ABB RAPID module: f527d16c.mod

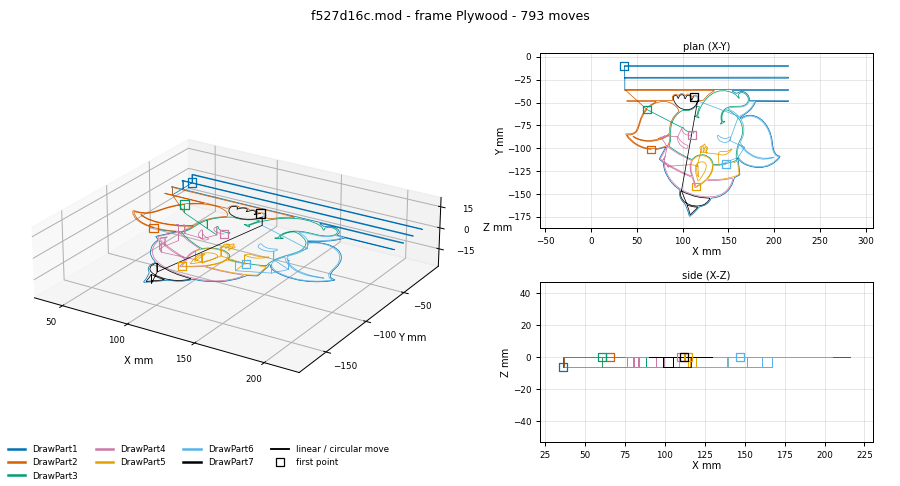
[picture p0: tool path of f527d16c.mod in frame Plywood, 793 of 795 moves have a stored position in this frame; points joined in program order, loops and branches not executed]
MODULE ImageDraw
  ! Generated 2026-10-07 09:04 for ABB GoFa CRB 15000-5/0.95: 26 strokes
  ! Page 250 x 180 mm. Work object Plywood: Z points DOWN, so pen-up is -Z and the tool uses orientation [1,0,0,0].
  ! Uses the tool 'tcp' and work object 'Plywood' that already exist on the controller.
  CONST robtarget pOrigin:=[[0,0,0],[1,0,0,0],[0,0,0,0],[9E9,9E9,9E9,9E9,9E9,9E9]];
  CONST jointtarget jHome:=[[0,0,0,0,30,0],[9E9,9E9,9E9,9E9,9E9,9E9]];
  CONST speeddata vTravel:=[250,200,5000,1000];

  PROC DrawImage()
    SingArea\Wrist;
    ConfL\Off;
    ConfJ\Off;
    MoveAbsJ jHome\NoEOffs,vTravel,fine,tcp;
    DrawPart1;
    DrawPart2;
    DrawPart3;
    DrawPart4;
    DrawPart5;
    DrawPart6;
    DrawPart7;
    MoveAbsJ jHome\NoEOffs,vTravel,fine,tcp;
  ENDPROC

  PROC DrawPart1()
    MoveL Offs(pOrigin,36.30,-10.13,-6.00),vTravel,z5,tcp\WObj:=Plywood;
    MoveL Offs(pOrigin,36.30,-10.13,-0.00),v60,z0,tcp\WObj:=Plywood;
    MoveL Offs(pOrigin,37.06,-9.56,-0.00),v40,z0,tcp\WObj:=Plywood;
    MoveL Offs(pOrigin,215.03,-9.56,-0.00),v40,z0,tcp\WObj:=Plywood;
    MoveL Offs(pOrigin,215.98,-9.94,-0.00),v40,z0,tcp\WObj:=Plywood;
    MoveL Offs(pOrigin,215.60,-10.51,-0.00),v40,z0,tcp\WObj:=Plywood;
    MoveL Offs(pOrigin,38.96,-10.70,-0.00),v40,z0,tcp\WObj:=Plywood;
    MoveL Offs(pOrigin,36.68,-10.51,-0.00),v40,z0,tcp\WObj:=Plywood;
    MoveL Offs(pOrigin,36.30,-10.13,-0.00),v40,fine,tcp\WObj:=Plywood;
    MoveL Offs(pOrigin,36.30,-10.13,-6.00),v60,z5,tcp\WObj:=Plywood;
    MoveL Offs(pOrigin,36.87,-22.47,-6.00),vTravel,z5,tcp\WObj:=Plywood;
    MoveL Offs(pOrigin,36.87,-22.47,-0.00),v60,z0,tcp\WObj:=Plywood;
    MoveL Offs(pOrigin,213.13,-22.28,-0.00),v40,z0,tcp\WObj:=Plywood;
    MoveL Offs(pOrigin,215.60,-22.47,-0.00),v40,z0,tcp\WObj:=Plywood;
    MoveL Offs(pOrigin,215.98,-22.85,-0.00),v40,z0,tcp\WObj:=Plywood;
    MoveL Offs(pOrigin,215.41,-23.42,-0.00),v40,z0,tcp\WObj:=Plywood;
    MoveL Offs(pOrigin,36.68,-23.42,-0.00),v40,z0,tcp\WObj:=Plywood;
    MoveL Offs(pOrigin,36.30,-23.04,-0.00),v40,z0,tcp\WObj:=Plywood;
    MoveL Offs(pOrigin,36.87,-22.47,-0.00),v40,fine,tcp\WObj:=Plywood;
    MoveL Offs(pOrigin,36.87,-22.47,-6.00),v60,z5,tcp\WObj:=Plywood;
    MoveL Offs(pOrigin,36.87,-35.77,-6.00),vTravel,z5,tcp\WObj:=Plywood;
    MoveL Offs(pOrigin,36.87,-35.77,-0.00),v60,z0,tcp\WObj:=Plywood;
    MoveL Offs(pOrigin,107.34,-35.96,-0.00),v40,z0,tcp\WObj:=Plywood;
    MoveL Offs(pOrigin,150.64,-35.58,-0.00),v40,z0,tcp\WObj:=Plywood;
    MoveL Offs(pOrigin,215.41,-35.77,-0.00),v40,z0,tcp\WObj:=Plywood;
    MoveL Offs(pOrigin,215.98,-36.15,-0.00),v40,z0,tcp\WObj:=Plywood;
    MoveL Offs(pOrigin,215.60,-36.72,-0.00),v40,z0,tcp\WObj:=Plywood;
    MoveL Offs(pOrigin,206.87,-36.91,-0.00),v40,z0,tcp\WObj:=Plywood;
    MoveL Offs(pOrigin,167.36,-36.72,-0.00),v40,z0,tcp\WObj:=Plywood;
    MoveL Offs(pOrigin,155.20,-36.91,-0.00),v40,z0,tcp\WObj:=Plywood;
    MoveL Offs(pOrigin,154.25,-37.16,-0.00),v40,z0,tcp\WObj:=Plywood;
    MoveL Offs(pOrigin,154.63,-37.73,-0.00),v40,z0,tcp\WObj:=Plywood;
    MoveL Offs(pOrigin,158.81,-40.01,-0.00),v40,z0,tcp\WObj:=Plywood;
    MoveL Offs(pOrigin,159.76,-39.44,-0.00),v40,z0,tcp\WObj:=Plywood;
    MoveL Offs(pOrigin,160.52,-39.44,-0.00),v40,z0,tcp\WObj:=Plywood;
    MoveL Offs(pOrigin,163.37,-37.86,-0.00),v40,z0,tcp\WObj:=Plywood;
    MoveL Offs(pOrigin,165.46,-37.86,-0.00),v40,z0,tcp\WObj:=Plywood;
    MoveL Offs(pOrigin,167.36,-38.37,-0.00),v40,z0,tcp\WObj:=Plywood;
    MoveL Offs(pOrigin,169.07,-39.25,-0.00),v40,z0,tcp\WObj:=Plywood;
    MoveL Offs(pOrigin,171.79,-42.23,-0.00),v40,z0,tcp\WObj:=Plywood;
    MoveL Offs(pOrigin,172.87,-44.70,-0.00),v40,z0,tcp\WObj:=Plywood;
    MoveL Offs(pOrigin,172.93,-47.55,-0.00),v40,z0,tcp\WObj:=Plywood;
    MoveL Offs(pOrigin,173.63,-47.93,-0.00),v40,z0,tcp\WObj:=Plywood;
    MoveL Offs(pOrigin,215.92,-48.12,-0.00),v40,z0,tcp\WObj:=Plywood;
    MoveL Offs(pOrigin,215.79,-48.62,-0.00),v40,z0,tcp\WObj:=Plywood;
    MoveL Offs(pOrigin,214.65,-48.88,-0.00),v40,z0,tcp\WObj:=Plywood;
    MoveL Offs(pOrigin,179.89,-48.81,-0.00),v40,z0,tcp\WObj:=Plywood;
    MoveL Offs(pOrigin,177.93,-53.06,-0.00),v40,z0,tcp\WObj:=Plywood;
    MoveL Offs(pOrigin,174.58,-57.61,-0.00),v40,z0,tcp\WObj:=Plywood;
    MoveL Offs(pOrigin,170.78,-61.03,-0.00),v40,z0,tcp\WObj:=Plywood;
    MoveL Offs(pOrigin,162.48,-66.54,-0.00),v40,z0,tcp\WObj:=Plywood;
    MoveL Offs(pOrigin,163.18,-67.49,-0.00),v40,z0,tcp\WObj:=Plywood;
    MoveL Offs(pOrigin,167.36,-65.15,-0.00),v40,z0,tcp\WObj:=Plywood;
    MoveL Offs(pOrigin,169.45,-64.45,-0.00),v40,z0,tcp\WObj:=Plywood;
    MoveL Offs(pOrigin,172.87,-63.88,-0.00),v40,z0,tcp\WObj:=Plywood;
    MoveL Offs(pOrigin,176.66,-64.07,-0.00),v40,z0,tcp\WObj:=Plywood;
    MoveL Offs(pOrigin,180.84,-65.34,-0.00),v40,z0,tcp\WObj:=Plywood;
    MoveL Offs(pOrigin,183.12,-66.48,-0.00),v40,z0,tcp\WObj:=Plywood;
    MoveL Offs(pOrigin,186.73,-69.01,-0.00),v40,z0,tcp\WObj:=Plywood;
    MoveL Offs(pOrigin,190.72,-73.38,-0.00),v40,z0,tcp\WObj:=Plywood;
    MoveL Offs(pOrigin,193.25,-77.37,-0.00),v40,z0,tcp\WObj:=Plywood;
    MoveL Offs(pOrigin,195.34,-81.74,-0.00),v40,z0,tcp\WObj:=Plywood;
    MoveL Offs(pOrigin,197.56,-89.34,-0.00),v40,z0,tcp\WObj:=Plywood;
    MoveL Offs(pOrigin,198.51,-97.31,-0.00),v40,z0,tcp\WObj:=Plywood;
    MoveL Offs(pOrigin,199.96,-103.20,-0.00),v40,z0,tcp\WObj:=Plywood;
    MoveL Offs(pOrigin,202.12,-106.62,-0.00),v40,z0,tcp\WObj:=Plywood;
    MoveL Offs(pOrigin,204.21,-108.01,-0.00),v40,z0,tcp\WObj:=Plywood;
    MoveL Offs(pOrigin,206.30,-108.58,-0.00),v40,z0,tcp\WObj:=Plywood;
    MoveL Offs(pOrigin,206.36,-109.47,-0.00),v40,z0,tcp\WObj:=Plywood;
    MoveL Offs(pOrigin,203.07,-113.46,-0.00),v40,z0,tcp\WObj:=Plywood;
    MoveL Offs(pOrigin,198.13,-117.13,-0.00),v40,z0,tcp\WObj:=Plywood;
    MoveL Offs(pOrigin,193.38,-119.41,-0.00),v40,z0,tcp\WObj:=Plywood;
    MoveL Offs(pOrigin,187.11,-120.87,-0.00),v40,z0,tcp\WObj:=Plywood;
    MoveL Offs(pOrigin,180.27,-120.87,-0.00),v40,z0,tcp\WObj:=Plywood;
    MoveL Offs(pOrigin,176.28,-120.30,-0.00),v40,z0,tcp\WObj:=Plywood;
    MoveL Offs(pOrigin,171.16,-118.84,-0.00),v40,z0,tcp\WObj:=Plywood;
    MoveL Offs(pOrigin,167.36,-117.13,-0.00),v40,z0,tcp\WObj:=Plywood;
    MoveL Offs(pOrigin,164.89,-115.55,-0.00),v40,z0,tcp\WObj:=Plywood;
    MoveL Offs(pOrigin,162.42,-113.27,-0.00),v40,z0,tcp\WObj:=Plywood;
    MoveL Offs(pOrigin,160.52,-110.61,-0.00),v40,z0,tcp\WObj:=Plywood;
    MoveL Offs(pOrigin,160.14,-110.48,-0.00),v40,z0,tcp\WObj:=Plywood;
    MoveL Offs(pOrigin,159.95,-111.37,-0.00),v40,z0,tcp\WObj:=Plywood;
    MoveL Offs(pOrigin,160.90,-113.84,-0.00),v40,z0,tcp\WObj:=Plywood;
    MoveL Offs(pOrigin,162.61,-128.46,-0.00),v40,z0,tcp\WObj:=Plywood;
    MoveL Offs(pOrigin,162.23,-129.22,-0.00),v40,z0,tcp\WObj:=Plywood;
    MoveL Offs(pOrigin,156.72,-132.07,-0.00),v40,z0,tcp\WObj:=Plywood;
    MoveL Offs(pOrigin,154.12,-139.67,-0.00),v40,z0,tcp\WObj:=Plywood;
    MoveL Offs(pOrigin,150.26,-145.75,-0.00),v40,z0,tcp\WObj:=Plywood;
    MoveL Offs(pOrigin,147.03,-148.79,-0.00),v40,z0,tcp\WObj:=Plywood;
    MoveL Offs(pOrigin,141.53,-152.14,-0.00),v40,z0,tcp\WObj:=Plywood;
    MoveL Offs(pOrigin,136.78,-153.73,-0.00),v40,z0,tcp\WObj:=Plywood;
    MoveL Offs(pOrigin,131.27,-154.55,-0.00),v40,z0,tcp\WObj:=Plywood;
    MoveL Offs(pOrigin,129.94,-157.15,-0.00),v40,z0,tcp\WObj:=Plywood;
    MoveL Offs(pOrigin,127.28,-160.18,-0.00),v40,z0,tcp\WObj:=Plywood;
    MoveL Offs(pOrigin,124.24,-162.21,-0.00),v40,z0,tcp\WObj:=Plywood;
    MoveL Offs(pOrigin,118.35,-164.17,-0.00),v40,z0,tcp\WObj:=Plywood;
    MoveL Offs(pOrigin,111.51,-171.39,-0.00),v40,z0,tcp\WObj:=Plywood;
    MoveL Offs(pOrigin,107.91,-174.37,-0.00),v40,z0,tcp\WObj:=Plywood;
    MoveL Offs(pOrigin,107.27,-173.86,-0.00),v40,z0,tcp\WObj:=Plywood;
    MoveL Offs(pOrigin,105.88,-168.92,-0.00),v40,z0,tcp\WObj:=Plywood;
    MoveL Offs(pOrigin,103.09,-161.89,-0.00),v40,z0,tcp\WObj:=Plywood;
    MoveL Offs(pOrigin,102.21,-160.37,-0.00),v40,z0,tcp\WObj:=Plywood;
    MoveL Offs(pOrigin,99.17,-156.96,-0.00),v40,z0,tcp\WObj:=Plywood;
    MoveL Offs(pOrigin,97.58,-154.11,-0.00),v40,z0,tcp\WObj:=Plywood;
    MoveL Offs(pOrigin,96.70,-150.88,-0.00),v40,z0,tcp\WObj:=Plywood;
    MoveL Offs(pOrigin,96.70,-148.41,-0.00),v40,z0,tcp\WObj:=Plywood;
    MoveL Offs(pOrigin,97.20,-145.75,-0.00),v40,z0,tcp\WObj:=Plywood;
    MoveL Offs(pOrigin,91.95,-141.57,-0.00),v40,z0,tcp\WObj:=Plywood;
    MoveL Offs(pOrigin,88.15,-137.77,-0.00),v40,z0,tcp\WObj:=Plywood;
    MoveL Offs(pOrigin,85.30,-133.97,-0.00),v40,z0,tcp\WObj:=Plywood;
    MoveL Offs(pOrigin,81.82,-127.70,-0.00),v40,z0,tcp\WObj:=Plywood;
    MoveL Offs(pOrigin,80.49,-124.28,-0.00),v40,z0,tcp\WObj:=Plywood;
    MoveL Offs(pOrigin,79.41,-120.11,-0.00),v40,z0,tcp\WObj:=Plywood;
    MoveL Offs(pOrigin,78.91,-115.55,-0.00),v40,z0,tcp\WObj:=Plywood;
    MoveL Offs(pOrigin,74.73,-112.13,-0.00),v40,z0,tcp\WObj:=Plywood;
    MoveL Offs(pOrigin,75.17,-110.42,-0.00),v40,z0,tcp\WObj:=Plywood;
    MoveL Offs(pOrigin,81.63,-98.83,-0.00),v40,z0,tcp\WObj:=Plywood;
    MoveL Offs(pOrigin,81.12,-98.64,-0.00),v40,z0,tcp\WObj:=Plywood;
    MoveL Offs(pOrigin,75.04,-100.54,-0.00),v40,z0,tcp\WObj:=Plywood;
    MoveL Offs(pOrigin,70.30,-101.30,-0.00),v40,z0,tcp\WObj:=Plywood;
  ENDPROC

  PROC DrawPart2()
    MoveL Offs(pOrigin,65.55,-101.30,-0.00),v40,z0,tcp\WObj:=Plywood;
    MoveL Offs(pOrigin,57.95,-99.97,-0.00),v40,z0,tcp\WObj:=Plywood;
    MoveL Offs(pOrigin,51.68,-97.57,-0.00),v40,z0,tcp\WObj:=Plywood;
    MoveL Offs(pOrigin,46.17,-94.08,-0.00),v40,z0,tcp\WObj:=Plywood;
    MoveL Offs(pOrigin,41.23,-89.53,-0.00),v40,z0,tcp\WObj:=Plywood;
    MoveL Offs(pOrigin,37.94,-84.97,-0.00),v40,z0,tcp\WObj:=Plywood;
    MoveL Offs(pOrigin,38.39,-84.21,-0.00),v40,z0,tcp\WObj:=Plywood;
    MoveL Offs(pOrigin,43.13,-84.21,-0.00),v40,z0,tcp\WObj:=Plywood;
    MoveL Offs(pOrigin,46.36,-83.32,-0.00),v40,z0,tcp\WObj:=Plywood;
    MoveL Offs(pOrigin,47.50,-82.69,-0.00),v40,z0,tcp\WObj:=Plywood;
    MoveL Offs(pOrigin,49.21,-80.98,-0.00),v40,z0,tcp\WObj:=Plywood;
    MoveL Offs(pOrigin,51.18,-76.80,-0.00),v40,z0,tcp\WObj:=Plywood;
    MoveL Offs(pOrigin,54.28,-66.92,-0.00),v40,z0,tcp\WObj:=Plywood;
    MoveL Offs(pOrigin,56.56,-62.17,-0.00),v40,z0,tcp\WObj:=Plywood;
    MoveL Offs(pOrigin,58.14,-59.70,-0.00),v40,z0,tcp\WObj:=Plywood;
    MoveL Offs(pOrigin,61.56,-55.53,-0.00),v40,z0,tcp\WObj:=Plywood;
    MoveL Offs(pOrigin,64.60,-52.87,-0.00),v40,z0,tcp\WObj:=Plywood;
    MoveL Offs(pOrigin,71.12,-49.07,-0.00),v40,z0,tcp\WObj:=Plywood;
    MoveL Offs(pOrigin,70.68,-48.69,-0.00),v40,z0,tcp\WObj:=Plywood;
    MoveL Offs(pOrigin,39.34,-48.69,-0.00),v40,z0,tcp\WObj:=Plywood;
    MoveL Offs(pOrigin,38.96,-48.31,-0.00),v40,z0,tcp\WObj:=Plywood;
    MoveL Offs(pOrigin,39.15,-47.99,-0.00),v40,z0,tcp\WObj:=Plywood;
    MoveL Offs(pOrigin,88.72,-47.93,-0.00),v40,z0,tcp\WObj:=Plywood;
    MoveL Offs(pOrigin,89.29,-47.36,-0.00),v40,z0,tcp\WObj:=Plywood;
    MoveL Offs(pOrigin,88.72,-43.75,-0.00),v40,z0,tcp\WObj:=Plywood;
    MoveL Offs(pOrigin,90.05,-41.85,-0.00),v40,z0,tcp\WObj:=Plywood;
    MoveL Offs(pOrigin,91.95,-40.96,-0.00),v40,z0,tcp\WObj:=Plywood;
    MoveL Offs(pOrigin,93.66,-41.09,-0.00),v40,z0,tcp\WObj:=Plywood;
    MoveL Offs(pOrigin,95.37,-42.29,-0.00),v40,z0,tcp\WObj:=Plywood;
    MoveL Offs(pOrigin,97.46,-40.65,-0.00),v40,z0,tcp\WObj:=Plywood;
    MoveL Offs(pOrigin,98.41,-40.33,-0.00),v40,z0,tcp\WObj:=Plywood;
    MoveL Offs(pOrigin,100.88,-40.65,-0.00),v40,z0,tcp\WObj:=Plywood;
    MoveL Offs(pOrigin,102.97,-42.55,-0.00),v40,z0,tcp\WObj:=Plywood;
    MoveL Offs(pOrigin,104.68,-41.15,-0.00),v40,z0,tcp\WObj:=Plywood;
    MoveL Offs(pOrigin,105.82,-40.77,-0.00),v40,z0,tcp\WObj:=Plywood;
    MoveL Offs(pOrigin,107.15,-40.90,-0.00),v40,z0,tcp\WObj:=Plywood;
    MoveL Offs(pOrigin,109.04,-42.04,-0.00),v40,z0,tcp\WObj:=Plywood;
    MoveL Offs(pOrigin,110.37,-43.81,-0.00),v40,z0,tcp\WObj:=Plywood;
    MoveL Offs(pOrigin,112.08,-42.36,-0.00),v40,z0,tcp\WObj:=Plywood;
    MoveL Offs(pOrigin,114.36,-42.04,-0.00),v40,z0,tcp\WObj:=Plywood;
    MoveL Offs(pOrigin,116.07,-42.99,-0.00),v40,z0,tcp\WObj:=Plywood;
    MoveL Offs(pOrigin,116.96,-44.13,-0.00),v40,z0,tcp\WObj:=Plywood;
    MoveL Offs(pOrigin,117.40,-45.27,-0.00),v40,z0,tcp\WObj:=Plywood;
    MoveL Offs(pOrigin,117.59,-47.67,-0.00),v40,z0,tcp\WObj:=Plywood;
    MoveL Offs(pOrigin,118.35,-47.93,-0.00),v40,z0,tcp\WObj:=Plywood;
    MoveL Offs(pOrigin,122.34,-47.74,-0.00),v40,z0,tcp\WObj:=Plywood;
    MoveL Offs(pOrigin,128.23,-41.34,-0.00),v40,z0,tcp\WObj:=Plywood;
    MoveL Offs(pOrigin,133.55,-37.73,-0.00),v40,z0,tcp\WObj:=Plywood;
    MoveL Offs(pOrigin,134.75,-37.29,-0.00),v40,z0,tcp\WObj:=Plywood;
    MoveL Offs(pOrigin,134.31,-36.91,-0.00),v40,z0,tcp\WObj:=Plywood;
    MoveL Offs(pOrigin,125.76,-36.72,-0.00),v40,z0,tcp\WObj:=Plywood;
    MoveL Offs(pOrigin,41.61,-36.91,-0.00),v40,z0,tcp\WObj:=Plywood;
    MoveL Offs(pOrigin,36.87,-36.72,-0.00),v40,z0,tcp\WObj:=Plywood;
    MoveL Offs(pOrigin,36.36,-36.34,-0.00),v40,z0,tcp\WObj:=Plywood;
    MoveL Offs(pOrigin,36.87,-35.77,-0.00),v40,fine,tcp\WObj:=Plywood;
    MoveL Offs(pOrigin,36.87,-35.77,-6.00),v60,z5,tcp\WObj:=Plywood;
    MoveL Offs(pOrigin,60.99,-57.61,-6.00),vTravel,z5,tcp\WObj:=Plywood;
    MoveL Offs(pOrigin,60.99,-57.61,-0.00),v60,z0,tcp\WObj:=Plywood;
    MoveL Offs(pOrigin,58.08,-61.60,-0.00),v40,z0,tcp\WObj:=Plywood;
    MoveL Offs(pOrigin,54.85,-68.25,-0.00),v40,z0,tcp\WObj:=Plywood;
    MoveL Offs(pOrigin,51.55,-78.70,-0.00),v40,z0,tcp\WObj:=Plywood;
    MoveL Offs(pOrigin,49.59,-82.12,-0.00),v40,z0,tcp\WObj:=Plywood;
    MoveL Offs(pOrigin,47.69,-83.76,-0.00),v40,z0,tcp\WObj:=Plywood;
    MoveL Offs(pOrigin,45.79,-84.65,-0.00),v40,z0,tcp\WObj:=Plywood;
    MoveL Offs(pOrigin,42.75,-85.35,-0.00),v40,z0,tcp\WObj:=Plywood;
    MoveL Offs(pOrigin,39.72,-85.41,-0.00),v40,z0,tcp\WObj:=Plywood;
    MoveL Offs(pOrigin,39.65,-85.92,-0.00),v40,z0,tcp\WObj:=Plywood;
    MoveL Offs(pOrigin,41.04,-87.82,-0.00),v40,z0,tcp\WObj:=Plywood;
    MoveL Offs(pOrigin,46.74,-93.32,-0.00),v40,z0,tcp\WObj:=Plywood;
    MoveL Offs(pOrigin,50.54,-95.86,-0.00),v40,z0,tcp\WObj:=Plywood;
    MoveL Offs(pOrigin,55.29,-98.14,-0.00),v40,z0,tcp\WObj:=Plywood;
    MoveL Offs(pOrigin,60.04,-99.59,-0.00),v40,z0,tcp\WObj:=Plywood;
    MoveL Offs(pOrigin,67.07,-100.54,-0.00),v40,z0,tcp\WObj:=Plywood;
    MoveL Offs(pOrigin,72.77,-100.16,-0.00),v40,z0,tcp\WObj:=Plywood;
    MoveL Offs(pOrigin,77.13,-99.21,-0.00),v40,z0,tcp\WObj:=Plywood;
    MoveL Offs(pOrigin,83.97,-96.68,-0.00),v40,z0,tcp\WObj:=Plywood;
    MoveL Offs(pOrigin,84.99,-94.84,-0.00),v40,z0,tcp\WObj:=Plywood;
    MoveL Offs(pOrigin,86.06,-90.66,-0.00),v40,z0,tcp\WObj:=Plywood;
    MoveL Offs(pOrigin,86.25,-85.35,-0.00),v40,z0,tcp\WObj:=Plywood;
    MoveL Offs(pOrigin,85.87,-84.97,-0.00),v40,z0,tcp\WObj:=Plywood;
    MoveL Offs(pOrigin,81.69,-87.88,-0.00),v40,z0,tcp\WObj:=Plywood;
    MoveL Offs(pOrigin,77.70,-89.78,-0.00),v40,z0,tcp\WObj:=Plywood;
    MoveL Offs(pOrigin,72.01,-91.42,-0.00),v40,z0,tcp\WObj:=Plywood;
    MoveL Offs(pOrigin,65.74,-92.37,-0.00),v40,z0,tcp\WObj:=Plywood;
    MoveL Offs(pOrigin,60.42,-92.37,-0.00),v40,z0,tcp\WObj:=Plywood;
    MoveL Offs(pOrigin,54.72,-91.42,-0.00),v40,z0,tcp\WObj:=Plywood;
    MoveL Offs(pOrigin,48.64,-89.08,-0.00),v40,z0,tcp\WObj:=Plywood;
    MoveL Offs(pOrigin,46.17,-87.56,-0.00),v40,z0,tcp\WObj:=Plywood;
    MoveL Offs(pOrigin,45.86,-86.93,-0.00),v40,z0,tcp\WObj:=Plywood;
    MoveL Offs(pOrigin,46.36,-86.93,-0.00),v40,z0,tcp\WObj:=Plywood;
    MoveL Offs(pOrigin,49.97,-89.02,-0.00),v40,z0,tcp\WObj:=Plywood;
    MoveL Offs(pOrigin,54.15,-90.47,-0.00),v40,z0,tcp\WObj:=Plywood;
    MoveL Offs(pOrigin,59.66,-91.42,-0.00),v40,z0,tcp\WObj:=Plywood;
    MoveL Offs(pOrigin,65.17,-91.42,-0.00),v40,z0,tcp\WObj:=Plywood;
    MoveL Offs(pOrigin,71.82,-90.47,-0.00),v40,z0,tcp\WObj:=Plywood;
    MoveL Offs(pOrigin,72.96,-89.72,-0.00),v40,z0,tcp\WObj:=Plywood;
    MoveL Offs(pOrigin,73.72,-89.84,-0.00),v40,z0,tcp\WObj:=Plywood;
    MoveL Offs(pOrigin,73.65,-89.34,-0.00),v40,z0,tcp\WObj:=Plywood;
    MoveL Offs(pOrigin,75.04,-89.53,-0.00),v40,z0,tcp\WObj:=Plywood;
    MoveL Offs(pOrigin,78.27,-88.45,-0.00),v40,z0,tcp\WObj:=Plywood;
    MoveL Offs(pOrigin,83.59,-85.54,-0.00),v40,z0,tcp\WObj:=Plywood;
    MoveL Offs(pOrigin,85.81,-83.07,-0.00),v40,z0,tcp\WObj:=Plywood;
    MoveL Offs(pOrigin,86.06,-82.31,-0.00),v40,z0,tcp\WObj:=Plywood;
    MoveL Offs(pOrigin,85.87,-77.94,-0.00),v40,z0,tcp\WObj:=Plywood;
    MoveL Offs(pOrigin,86.82,-73.00,-0.00),v40,z0,tcp\WObj:=Plywood;
    MoveL Offs(pOrigin,87.90,-70.15,-0.00),v40,z0,tcp\WObj:=Plywood;
    MoveL Offs(pOrigin,89.61,-66.92,-0.00),v40,z0,tcp\WObj:=Plywood;
    MoveL Offs(pOrigin,91.38,-64.45,-0.00),v40,z0,tcp\WObj:=Plywood;
    MoveL Offs(pOrigin,94.61,-60.84,-0.00),v40,z0,tcp\WObj:=Plywood;
    MoveL Offs(pOrigin,96.07,-59.89,-0.00),v40,z0,tcp\WObj:=Plywood;
    MoveL Offs(pOrigin,95.43,-57.80,-0.00),v40,z0,tcp\WObj:=Plywood;
    MoveL Offs(pOrigin,93.47,-54.96,-0.00),v40,z0,tcp\WObj:=Plywood;
    MoveL Offs(pOrigin,91.00,-52.68,-0.00),v40,z0,tcp\WObj:=Plywood;
    MoveL Offs(pOrigin,87.77,-50.71,-0.00),v40,z0,tcp\WObj:=Plywood;
    MoveL Offs(pOrigin,83.40,-49.26,-0.00),v40,z0,tcp\WObj:=Plywood;
    MoveL Offs(pOrigin,80.93,-48.88,-0.00),v40,z0,tcp\WObj:=Plywood;
    MoveL Offs(pOrigin,75.80,-49.07,-0.00),v40,z0,tcp\WObj:=Plywood;
    MoveL Offs(pOrigin,71.06,-50.33,-0.00),v40,z0,tcp\WObj:=Plywood;
    MoveL Offs(pOrigin,68.40,-51.60,-0.00),v40,z0,tcp\WObj:=Plywood;
    MoveL Offs(pOrigin,63.65,-54.96,-0.00),v40,z0,tcp\WObj:=Plywood;
  ENDPROC

  PROC DrawPart3()
    MoveL Offs(pOrigin,60.99,-57.61,-0.00),v40,fine,tcp\WObj:=Plywood;
    MoveL Offs(pOrigin,60.99,-57.61,-6.00),v60,z5,tcp\WObj:=Plywood;
    MoveL Offs(pOrigin,88.47,-71.86,-6.00),vTravel,z5,tcp\WObj:=Plywood;
    MoveL Offs(pOrigin,88.47,-71.86,-0.00),v60,z0,tcp\WObj:=Plywood;
    MoveL Offs(pOrigin,87.77,-74.14,-0.00),v40,z0,tcp\WObj:=Plywood;
    MoveL Offs(pOrigin,87.07,-78.51,-0.00),v40,z0,tcp\WObj:=Plywood;
    MoveL Offs(pOrigin,87.01,-90.66,-0.00),v40,z0,tcp\WObj:=Plywood;
    MoveL Offs(pOrigin,86.06,-94.84,-0.00),v40,z0,tcp\WObj:=Plywood;
    MoveL Offs(pOrigin,85.11,-97.31,-0.00),v40,z0,tcp\WObj:=Plywood;
    MoveL Offs(pOrigin,85.30,-97.69,-0.00),v40,z0,tcp\WObj:=Plywood;
    MoveL Offs(pOrigin,89.48,-100.92,-0.00),v40,z0,tcp\WObj:=Plywood;
    MoveL Offs(pOrigin,95.75,-104.97,-0.00),v40,z0,tcp\WObj:=Plywood;
    MoveL Offs(pOrigin,103.92,-109.53,-0.00),v40,z0,tcp\WObj:=Plywood;
    MoveL Offs(pOrigin,110.18,-112.32,-0.00),v40,z0,tcp\WObj:=Plywood;
    MoveL Offs(pOrigin,113.60,-109.28,-0.00),v40,z0,tcp\WObj:=Plywood;
    MoveL Offs(pOrigin,117.02,-107.57,-0.00),v40,z0,tcp\WObj:=Plywood;
    MoveL Offs(pOrigin,121.77,-107.00,-0.00),v40,z0,tcp\WObj:=Plywood;
    MoveL Offs(pOrigin,123.67,-107.19,-0.00),v40,z0,tcp\WObj:=Plywood;
    MoveL Offs(pOrigin,125.76,-107.89,-0.00),v40,z0,tcp\WObj:=Plywood;
    MoveL Offs(pOrigin,130.13,-110.61,-0.00),v40,z0,tcp\WObj:=Plywood;
    MoveL Offs(pOrigin,131.96,-113.08,-0.00),v40,z0,tcp\WObj:=Plywood;
    MoveL Offs(pOrigin,133.42,-117.26,-0.00),v40,z0,tcp\WObj:=Plywood;
    MoveL Offs(pOrigin,133.93,-117.64,-0.00),v40,z0,tcp\WObj:=Plywood;
    MoveL Offs(pOrigin,139.82,-117.64,-0.00),v40,z0,tcp\WObj:=Plywood;
    MoveL Offs(pOrigin,146.65,-116.69,-0.00),v40,z0,tcp\WObj:=Plywood;
    MoveL Offs(pOrigin,153.11,-115.36,-0.00),v40,z0,tcp\WObj:=Plywood;
    MoveL Offs(pOrigin,158.62,-113.33,-0.00),v40,z0,tcp\WObj:=Plywood;
    MoveL Offs(pOrigin,159.19,-112.70,-0.00),v40,z0,tcp\WObj:=Plywood;
    MoveL Offs(pOrigin,158.62,-109.09,-0.00),v40,z0,tcp\WObj:=Plywood;
    MoveL Offs(pOrigin,158.62,-106.62,-0.00),v40,z0,tcp\WObj:=Plywood;
    MoveL Offs(pOrigin,159.57,-99.78,-0.00),v40,z0,tcp\WObj:=Plywood;
    MoveL Offs(pOrigin,161.53,-93.89,-0.00),v40,z0,tcp\WObj:=Plywood;
    MoveL Offs(pOrigin,164.26,-88.20,-0.00),v40,z0,tcp\WObj:=Plywood;
    MoveL Offs(pOrigin,165.46,-83.45,-0.00),v40,z0,tcp\WObj:=Plywood;
    MoveL Offs(pOrigin,165.65,-79.46,-0.00),v40,z0,tcp\WObj:=Plywood;
    MoveL Offs(pOrigin,164.57,-73.76,-0.00),v40,z0,tcp\WObj:=Plywood;
    MoveL Offs(pOrigin,162.48,-69.20,-0.00),v40,z0,tcp\WObj:=Plywood;
    MoveL Offs(pOrigin,158.81,-64.64,-0.00),v40,z0,tcp\WObj:=Plywood;
    MoveL Offs(pOrigin,153.30,-60.40,-0.00),v40,z0,tcp\WObj:=Plywood;
    MoveL Offs(pOrigin,151.40,-59.26,-0.00),v40,z0,tcp\WObj:=Plywood;
    MoveL Offs(pOrigin,147.98,-57.99,-0.00),v40,z0,tcp\WObj:=Plywood;
    MoveL Offs(pOrigin,146.65,-58.12,-0.00),v40,z0,tcp\WObj:=Plywood;
    MoveL Offs(pOrigin,145.13,-59.51,-0.00),v40,z0,tcp\WObj:=Plywood;
    MoveL Offs(pOrigin,143.93,-61.41,-0.00),v40,z0,tcp\WObj:=Plywood;
    MoveL Offs(pOrigin,143.04,-64.64,-0.00),v40,z0,tcp\WObj:=Plywood;
    MoveL Offs(pOrigin,143.04,-68.25,-0.00),v40,z0,tcp\WObj:=Plywood;
    MoveL Offs(pOrigin,143.49,-70.34,-0.00),v40,z0,tcp\WObj:=Plywood;
    MoveL Offs(pOrigin,144.18,-70.97,-0.00),v40,z0,tcp\WObj:=Plywood;
    MoveL Offs(pOrigin,146.08,-70.34,-0.00),v40,z0,tcp\WObj:=Plywood;
    MoveL Offs(pOrigin,146.21,-70.91,-0.00),v40,z0,tcp\WObj:=Plywood;
    MoveL Offs(pOrigin,142.09,-73.44,-0.00),v40,z0,tcp\WObj:=Plywood;
    MoveL Offs(pOrigin,141.53,-73.51,-0.00),v40,z0,tcp\WObj:=Plywood;
    MoveL Offs(pOrigin,141.40,-73.00,-0.00),v40,z0,tcp\WObj:=Plywood;
    MoveL Offs(pOrigin,142.85,-71.48,-0.00),v40,z0,tcp\WObj:=Plywood;
    MoveL Offs(pOrigin,142.09,-68.44,-0.00),v40,z0,tcp\WObj:=Plywood;
    MoveL Offs(pOrigin,142.09,-64.26,-0.00),v40,z0,tcp\WObj:=Plywood;
    MoveL Offs(pOrigin,142.98,-61.22,-0.00),v40,z0,tcp\WObj:=Plywood;
    MoveL Offs(pOrigin,144.18,-59.13,-0.00),v40,z0,tcp\WObj:=Plywood;
    MoveL Offs(pOrigin,146.46,-56.85,-0.00),v40,z0,tcp\WObj:=Plywood;
    MoveL Offs(pOrigin,148.74,-55.59,-0.00),v40,z0,tcp\WObj:=Plywood;
    MoveL Offs(pOrigin,151.97,-54.58,-0.00),v40,z0,tcp\WObj:=Plywood;
    MoveL Offs(pOrigin,155.39,-54.20,-0.00),v40,z0,tcp\WObj:=Plywood;
    MoveL Offs(pOrigin,163.75,-54.01,-0.00),v40,z0,tcp\WObj:=Plywood;
    MoveL Offs(pOrigin,167.55,-52.99,-0.00),v40,z0,tcp\WObj:=Plywood;
    MoveL Offs(pOrigin,169.83,-51.54,-0.00),v40,z0,tcp\WObj:=Plywood;
    MoveL Offs(pOrigin,171.47,-49.07,-0.00),v40,z0,tcp\WObj:=Plywood;
    MoveL Offs(pOrigin,171.92,-46.60,-0.00),v40,z0,tcp\WObj:=Plywood;
    MoveL Offs(pOrigin,171.54,-44.70,-0.00),v40,z0,tcp\WObj:=Plywood;
    MoveL Offs(pOrigin,170.65,-42.80,-0.00),v40,z0,tcp\WObj:=Plywood;
    MoveL Offs(pOrigin,169.07,-40.90,-0.00),v40,z0,tcp\WObj:=Plywood;
    MoveL Offs(pOrigin,167.36,-39.82,-0.00),v40,z0,tcp\WObj:=Plywood;
    MoveL Offs(pOrigin,165.46,-39.19,-0.00),v40,z0,tcp\WObj:=Plywood;
    MoveL Offs(pOrigin,163.56,-39.19,-0.00),v40,z0,tcp\WObj:=Plywood;
    MoveL Offs(pOrigin,161.66,-40.33,-0.00),v40,z0,tcp\WObj:=Plywood;
    MoveL Offs(pOrigin,160.90,-42.04,-0.00),v40,z0,tcp\WObj:=Plywood;
    MoveL Offs(pOrigin,161.03,-42.99,-0.00),v40,z0,tcp\WObj:=Plywood;
    MoveL Offs(pOrigin,162.04,-44.89,-0.00),v40,z0,tcp\WObj:=Plywood;
    MoveL Offs(pOrigin,161.66,-45.46,-0.00),v40,z0,tcp\WObj:=Plywood;
    MoveL Offs(pOrigin,158.24,-41.66,-0.00),v40,z0,tcp\WObj:=Plywood;
    MoveL Offs(pOrigin,155.96,-40.08,-0.00),v40,z0,tcp\WObj:=Plywood;
    MoveL Offs(pOrigin,152.73,-38.56,-0.00),v40,z0,tcp\WObj:=Plywood;
    MoveL Offs(pOrigin,146.46,-37.10,-0.00),v40,z0,tcp\WObj:=Plywood;
    MoveL Offs(pOrigin,140.39,-37.29,-0.00),v40,z0,tcp\WObj:=Plywood;
    MoveL Offs(pOrigin,135.64,-38.75,-0.00),v40,z0,tcp\WObj:=Plywood;
    MoveL Offs(pOrigin,132.60,-40.27,-0.00),v40,z0,tcp\WObj:=Plywood;
    MoveL Offs(pOrigin,128.61,-43.18,-0.00),v40,z0,tcp\WObj:=Plywood;
    MoveL Offs(pOrigin,124.24,-47.93,-0.00),v40,z0,tcp\WObj:=Plywood;
    MoveL Offs(pOrigin,120.38,-53.82,-0.00),v40,z0,tcp\WObj:=Plywood;
    MoveL Offs(pOrigin,117.78,-59.70,-0.00),v40,z0,tcp\WObj:=Plywood;
    MoveL Offs(pOrigin,116.45,-65.02,-0.00),v40,z0,tcp\WObj:=Plywood;
    MoveL Offs(pOrigin,117.97,-66.16,-0.00),v40,z0,tcp\WObj:=Plywood;
    MoveL Offs(pOrigin,118.10,-66.67,-0.00),v40,z0,tcp\WObj:=Plywood;
    MoveL Offs(pOrigin,117.59,-66.73,-0.00),v40,z0,tcp\WObj:=Plywood;
    MoveL Offs(pOrigin,113.03,-65.02,-0.00),v40,z0,tcp\WObj:=Plywood;
    MoveL Offs(pOrigin,113.41,-64.64,-0.00),v40,z0,tcp\WObj:=Plywood;
    MoveL Offs(pOrigin,115.44,-64.64,-0.00),v40,z0,tcp\WObj:=Plywood;
    MoveL Offs(pOrigin,116.83,-59.13,-0.00),v40,z0,tcp\WObj:=Plywood;
    MoveL Offs(pOrigin,118.35,-54.96,-0.00),v40,z0,tcp\WObj:=Plywood;
    MoveL Offs(pOrigin,117.97,-54.26,-0.00),v40,z0,tcp\WObj:=Plywood;
    MoveL Offs(pOrigin,115.50,-54.20,-0.00),v40,z0,tcp\WObj:=Plywood;
    MoveL Offs(pOrigin,114.36,-54.51,-0.00),v40,z0,tcp\WObj:=Plywood;
    MoveL Offs(pOrigin,110.75,-57.17,-0.00),v40,z0,tcp\WObj:=Plywood;
    MoveL Offs(pOrigin,106.39,-58.75,-0.00),v40,z0,tcp\WObj:=Plywood;
    MoveL Offs(pOrigin,101.64,-58.75,-0.00),v40,z0,tcp\WObj:=Plywood;
    MoveL Offs(pOrigin,100.31,-58.37,-0.00),v40,z0,tcp\WObj:=Plywood;
    MoveL Offs(pOrigin,96.70,-60.65,-0.00),v40,z0,tcp\WObj:=Plywood;
    MoveL Offs(pOrigin,93.47,-63.50,-0.00),v40,z0,tcp\WObj:=Plywood;
    MoveL Offs(pOrigin,90.37,-67.68,-0.00),v40,z0,tcp\WObj:=Plywood;
    MoveL Offs(pOrigin,88.47,-71.86,-0.00),v40,fine,tcp\WObj:=Plywood;
    MoveL Offs(pOrigin,88.47,-71.86,-6.00),v60,z5,tcp\WObj:=Plywood;
    MoveL Offs(pOrigin,99.48,-77.37,-6.00),vTravel,z5,tcp\WObj:=Plywood;
    MoveL Offs(pOrigin,99.48,-77.37,-0.00),v60,z0,tcp\WObj:=Plywood;
    MoveL Offs(pOrigin,100.12,-76.86,-0.00),v40,z0,tcp\WObj:=Plywood;
    MoveL Offs(pOrigin,102.59,-79.84,-0.00),v40,z0,tcp\WObj:=Plywood;
    MoveL Offs(pOrigin,105.25,-81.42,-0.00),v40,z0,tcp\WObj:=Plywood;
    MoveL Offs(pOrigin,107.34,-82.12,-0.00),v40,z0,tcp\WObj:=Plywood;
    MoveL Offs(pOrigin,109.61,-82.12,-0.00),v40,z0,tcp\WObj:=Plywood;
    MoveL Offs(pOrigin,112.08,-81.23,-0.00),v40,z0,tcp\WObj:=Plywood;
    MoveL Offs(pOrigin,112.46,-82.12,-0.00),v40,z0,tcp\WObj:=Plywood;
    MoveL Offs(pOrigin,111.96,-83.45,-0.00),v40,z0,tcp\WObj:=Plywood;
  ENDPROC

  PROC DrawPart4()
    MoveL Offs(pOrigin,109.99,-85.22,-0.00),v40,z0,tcp\WObj:=Plywood;
    MoveL Offs(pOrigin,108.09,-85.73,-0.00),v40,z0,tcp\WObj:=Plywood;
    MoveL Offs(pOrigin,104.87,-85.35,-0.00),v40,z0,tcp\WObj:=Plywood;
    MoveL Offs(pOrigin,102.97,-84.65,-0.00),v40,z0,tcp\WObj:=Plywood;
    MoveL Offs(pOrigin,101.45,-83.64,-0.00),v40,z0,tcp\WObj:=Plywood;
    MoveL Offs(pOrigin,99.99,-81.74,-0.00),v40,z0,tcp\WObj:=Plywood;
    MoveL Offs(pOrigin,99.36,-80.03,-0.00),v40,z0,tcp\WObj:=Plywood;
    MoveL Offs(pOrigin,99.48,-77.37,-0.00),v40,fine,tcp\WObj:=Plywood;
    MoveL Offs(pOrigin,99.48,-77.37,-6.00),v60,z5,tcp\WObj:=Plywood;
    MoveL Offs(pOrigin,94.74,-87.25,-6.00),vTravel,z5,tcp\WObj:=Plywood;
    MoveL Offs(pOrigin,94.74,-87.25,-0.00),v60,z0,tcp\WObj:=Plywood;
    MoveL Offs(pOrigin,96.89,-90.85,-0.00),v40,z0,tcp\WObj:=Plywood;
    MoveL Offs(pOrigin,99.74,-93.70,-0.00),v40,z0,tcp\WObj:=Plywood;
    MoveL Offs(pOrigin,102.40,-95.48,-0.00),v40,z0,tcp\WObj:=Plywood;
    MoveL Offs(pOrigin,105.94,-97.00,-0.00),v40,z0,tcp\WObj:=Plywood;
    MoveL Offs(pOrigin,105.69,-98.64,-0.00),v40,z0,tcp\WObj:=Plywood;
    MoveL Offs(pOrigin,104.68,-100.23,-0.00),v40,z0,tcp\WObj:=Plywood;
    MoveL Offs(pOrigin,103.35,-100.04,-0.00),v40,z0,tcp\WObj:=Plywood;
    MoveL Offs(pOrigin,100.88,-98.96,-0.00),v40,z0,tcp\WObj:=Plywood;
    MoveL Offs(pOrigin,97.27,-96.17,-0.00),v40,z0,tcp\WObj:=Plywood;
    MoveL Offs(pOrigin,95.31,-92.75,-0.00),v40,z0,tcp\WObj:=Plywood;
    MoveL Offs(pOrigin,94.04,-88.01,-0.00),v40,z0,tcp\WObj:=Plywood;
    MoveL Offs(pOrigin,94.23,-87.12,-0.00),v40,z0,tcp\WObj:=Plywood;
    MoveL Offs(pOrigin,94.74,-87.25,-0.00),v40,fine,tcp\WObj:=Plywood;
    MoveL Offs(pOrigin,94.74,-87.25,-6.00),v60,z5,tcp\WObj:=Plywood;
    MoveL Offs(pOrigin,80.43,-86.55,-6.00),vTravel,z5,tcp\WObj:=Plywood;
    MoveL Offs(pOrigin,80.43,-86.55,-0.00),v60,z0,tcp\WObj:=Plywood;
    MoveL Offs(pOrigin,79.41,-87.06,-0.00),v40,z0,tcp\WObj:=Plywood;
    MoveL Offs(pOrigin,79.79,-86.61,-0.00),v40,z0,tcp\WObj:=Plywood;
    MoveL Offs(pOrigin,80.43,-86.55,-0.00),v40,fine,tcp\WObj:=Plywood;
    MoveL Offs(pOrigin,80.43,-86.55,-6.00),v60,z5,tcp\WObj:=Plywood;
    MoveL Offs(pOrigin,76.44,-88.01,-6.00),vTravel,z5,tcp\WObj:=Plywood;
    MoveL Offs(pOrigin,76.44,-88.01,-0.00),v60,z0,tcp\WObj:=Plywood;
    MoveL Offs(pOrigin,76.18,-88.45,-0.00),v40,z0,tcp\WObj:=Plywood;
    MoveL Offs(pOrigin,74.92,-88.64,-0.00),v40,z0,tcp\WObj:=Plywood;
    MoveL Offs(pOrigin,75.80,-87.88,-0.00),v40,z0,tcp\WObj:=Plywood;
    MoveL Offs(pOrigin,76.44,-88.01,-0.00),v40,fine,tcp\WObj:=Plywood;
    MoveL Offs(pOrigin,76.44,-88.01,-6.00),v60,z5,tcp\WObj:=Plywood;
    MoveL Offs(pOrigin,83.21,-98.26,-6.00),vTravel,z5,tcp\WObj:=Plywood;
    MoveL Offs(pOrigin,83.21,-98.26,-0.00),v60,z0,tcp\WObj:=Plywood;
    MoveL Offs(pOrigin,75.80,-111.37,-0.00),v40,z0,tcp\WObj:=Plywood;
    MoveL Offs(pOrigin,75.99,-111.94,-0.00),v40,z0,tcp\WObj:=Plywood;
    MoveL Offs(pOrigin,82.64,-116.56,-0.00),v40,z0,tcp\WObj:=Plywood;
    MoveL Offs(pOrigin,90.62,-121.37,-0.00),v40,z0,tcp\WObj:=Plywood;
    MoveL Offs(pOrigin,101.83,-127.07,-0.00),v40,z0,tcp\WObj:=Plywood;
    MoveL Offs(pOrigin,109.80,-130.30,-0.00),v40,z0,tcp\WObj:=Plywood;
    MoveL Offs(pOrigin,109.99,-129.98,-0.00),v40,z0,tcp\WObj:=Plywood;
    MoveL Offs(pOrigin,108.85,-125.80,-0.00),v40,z0,tcp\WObj:=Plywood;
    MoveL Offs(pOrigin,108.28,-122.20,-0.00),v40,z0,tcp\WObj:=Plywood;
    MoveL Offs(pOrigin,108.28,-118.40,-0.00),v40,z0,tcp\WObj:=Plywood;
    MoveL Offs(pOrigin,109.61,-113.65,-0.00),v40,z0,tcp\WObj:=Plywood;
    MoveL Offs(pOrigin,109.42,-113.27,-0.00),v40,z0,tcp\WObj:=Plywood;
    MoveL Offs(pOrigin,95.75,-106.30,-0.00),v40,z0,tcp\WObj:=Plywood;
    MoveL Offs(pOrigin,86.63,-100.35,-0.00),v40,z0,tcp\WObj:=Plywood;
    MoveL Offs(pOrigin,83.97,-98.14,-0.00),v40,z0,tcp\WObj:=Plywood;
    MoveL Offs(pOrigin,83.21,-98.26,-0.00),v40,fine,tcp\WObj:=Plywood;
    MoveL Offs(pOrigin,83.21,-98.26,-6.00),v60,z5,tcp\WObj:=Plywood;
    MoveL Offs(pOrigin,80.74,-109.66,-6.00),vTravel,z5,tcp\WObj:=Plywood;
    MoveL Offs(pOrigin,80.74,-109.66,-0.00),v60,z0,tcp\WObj:=Plywood;
    MoveL Offs(pOrigin,81.31,-108.71,-0.00),v40,z0,tcp\WObj:=Plywood;
    MoveL Offs(pOrigin,80.74,-109.66,-0.00),v40,z0,tcp\WObj:=Plywood;
    MoveL Offs(pOrigin,80.11,-110.29,-0.00),v40,z0,tcp\WObj:=Plywood;
    MoveL Offs(pOrigin,80.30,-111.75,-0.00),v40,z0,tcp\WObj:=Plywood;
    MoveL Offs(pOrigin,79.41,-111.81,-0.00),v40,z0,tcp\WObj:=Plywood;
    MoveL Offs(pOrigin,78.97,-112.64,-0.00),v40,z0,tcp\WObj:=Plywood;
    MoveL Offs(pOrigin,78.46,-112.76,-0.00),v40,z0,tcp\WObj:=Plywood;
    MoveL Offs(pOrigin,80.11,-110.29,-0.00),v40,fine,tcp\WObj:=Plywood;
    MoveL Offs(pOrigin,80.11,-110.29,-6.00),v60,z5,tcp\WObj:=Plywood;
    MoveL Offs(pOrigin,80.55,-116.50,-6.00),vTravel,z5,tcp\WObj:=Plywood;
    MoveL Offs(pOrigin,80.55,-116.50,-0.00),v60,z0,tcp\WObj:=Plywood;
    MoveL Offs(pOrigin,80.17,-116.88,-0.00),v40,z0,tcp\WObj:=Plywood;
    MoveL Offs(pOrigin,80.17,-118.40,-0.00),v40,z0,tcp\WObj:=Plywood;
    MoveL Offs(pOrigin,81.12,-122.77,-0.00),v40,z0,tcp\WObj:=Plywood;
    MoveL Offs(pOrigin,84.10,-129.79,-0.00),v40,z0,tcp\WObj:=Plywood;
    MoveL Offs(pOrigin,87.77,-135.30,-0.00),v40,z0,tcp\WObj:=Plywood;
    MoveL Offs(pOrigin,92.33,-140.24,-0.00),v40,z0,tcp\WObj:=Plywood;
    MoveL Offs(pOrigin,95.75,-143.09,-0.00),v40,z0,tcp\WObj:=Plywood;
    MoveL Offs(pOrigin,98.98,-145.24,-0.00),v40,z0,tcp\WObj:=Plywood;
    MoveL Offs(pOrigin,103.35,-147.52,-0.00),v40,z0,tcp\WObj:=Plywood;
    MoveL Offs(pOrigin,112.27,-150.88,-0.00),v40,z0,tcp\WObj:=Plywood;
    MoveL Offs(pOrigin,117.02,-152.02,-0.00),v40,z0,tcp\WObj:=Plywood;
    MoveL Offs(pOrigin,124.24,-152.97,-0.00),v40,z0,tcp\WObj:=Plywood;
    MoveL Offs(pOrigin,129.75,-153.16,-0.00),v40,z0,tcp\WObj:=Plywood;
    MoveL Offs(pOrigin,132.22,-152.59,-0.00),v40,z0,tcp\WObj:=Plywood;
    MoveL Offs(pOrigin,135.64,-152.59,-0.00),v40,z0,tcp\WObj:=Plywood;
    MoveL Offs(pOrigin,141.15,-150.75,-0.00),v40,z0,tcp\WObj:=Plywood;
    MoveL Offs(pOrigin,143.99,-149.29,-0.00),v40,z0,tcp\WObj:=Plywood;
    MoveL Offs(pOrigin,146.84,-147.27,-0.00),v40,z0,tcp\WObj:=Plywood;
    MoveL Offs(pOrigin,149.31,-144.80,-0.00),v40,z0,tcp\WObj:=Plywood;
    MoveL Offs(pOrigin,151.85,-141.38,-0.00),v40,z0,tcp\WObj:=Plywood;
    MoveL Offs(pOrigin,154.19,-136.44,-0.00),v40,z0,tcp\WObj:=Plywood;
    MoveL Offs(pOrigin,154.82,-134.35,-0.00),v40,z0,tcp\WObj:=Plywood;
    MoveL Offs(pOrigin,154.44,-133.09,-0.00),v40,z0,tcp\WObj:=Plywood;
    MoveL Offs(pOrigin,152.92,-133.02,-0.00),v40,z0,tcp\WObj:=Plywood;
    MoveL Offs(pOrigin,146.84,-134.16,-0.00),v40,z0,tcp\WObj:=Plywood;
    MoveL Offs(pOrigin,138.11,-135.11,-0.00),v40,z0,tcp\WObj:=Plywood;
    MoveL Offs(pOrigin,129.37,-135.11,-0.00),v40,z0,tcp\WObj:=Plywood;
    MoveL Offs(pOrigin,126.14,-134.73,-0.00),v40,z0,tcp\WObj:=Plywood;
    MoveL Offs(pOrigin,121.20,-138.72,-0.00),v40,z0,tcp\WObj:=Plywood;
    MoveL Offs(pOrigin,113.79,-143.09,-0.00),v40,z0,tcp\WObj:=Plywood;
    MoveL Offs(pOrigin,113.41,-142.71,-0.00),v40,z0,tcp\WObj:=Plywood;
    MoveL Offs(pOrigin,112.65,-137.77,-0.00),v40,z0,tcp\WObj:=Plywood;
    MoveL Offs(pOrigin,110.56,-131.88,-0.00),v40,z0,tcp\WObj:=Plywood;
    MoveL Offs(pOrigin,97.27,-126.06,-0.00),v40,z0,tcp\WObj:=Plywood;
    MoveL Offs(pOrigin,85.30,-119.66,-0.00),v40,z0,tcp\WObj:=Plywood;
    MoveL Offs(pOrigin,81.31,-116.81,-0.00),v40,z0,tcp\WObj:=Plywood;
    MoveL Offs(pOrigin,80.55,-116.50,-0.00),v40,fine,tcp\WObj:=Plywood;
    MoveL Offs(pOrigin,80.55,-116.50,-6.00),v60,z5,tcp\WObj:=Plywood;
    MoveL Offs(pOrigin,83.97,-119.66,-6.00),vTravel,z5,tcp\WObj:=Plywood;
    MoveL Offs(pOrigin,83.97,-119.66,-0.00),v60,z0,tcp\WObj:=Plywood;
    MoveL Offs(pOrigin,84.48,-120.80,-0.00),v40,z0,tcp\WObj:=Plywood;
    MoveL Offs(pOrigin,84.04,-120.49,-0.00),v40,z0,tcp\WObj:=Plywood;
    MoveL Offs(pOrigin,83.97,-119.66,-0.00),v40,fine,tcp\WObj:=Plywood;
    MoveL Offs(pOrigin,83.97,-119.66,-6.00),v60,z5,tcp\WObj:=Plywood;
    MoveL Offs(pOrigin,109.23,-117.83,-6.00),vTravel,z5,tcp\WObj:=Plywood;
    MoveL Offs(pOrigin,109.23,-117.83,-0.00),v60,z0,tcp\WObj:=Plywood;
    MoveL Offs(pOrigin,109.23,-123.53,-0.00),v40,z0,tcp\WObj:=Plywood;
    MoveL Offs(pOrigin,109.61,-125.61,-0.00),v40,z0,tcp\WObj:=Plywood;
    MoveL Offs(pOrigin,113.03,-136.25,-0.00),v40,z0,tcp\WObj:=Plywood;
    MoveL Offs(pOrigin,114.17,-141.00,-0.00),v40,z0,tcp\WObj:=Plywood;
  ENDPROC

  PROC DrawPart5()
    MoveL Offs(pOrigin,114.74,-141.76,-0.00),v40,z0,tcp\WObj:=Plywood;
    MoveL Offs(pOrigin,119.49,-138.91,-0.00),v40,z0,tcp\WObj:=Plywood;
    MoveL Offs(pOrigin,125.38,-134.35,-0.00),v40,z0,tcp\WObj:=Plywood;
    MoveL Offs(pOrigin,128.23,-131.12,-0.00),v40,z0,tcp\WObj:=Plywood;
    MoveL Offs(pOrigin,129.62,-129.03,-0.00),v40,z0,tcp\WObj:=Plywood;
    MoveL Offs(pOrigin,131.65,-124.85,-0.00),v40,z0,tcp\WObj:=Plywood;
    MoveL Offs(pOrigin,132.60,-121.06,-0.00),v40,z0,tcp\WObj:=Plywood;
    MoveL Offs(pOrigin,132.60,-117.83,-0.00),v40,z0,tcp\WObj:=Plywood;
    MoveL Offs(pOrigin,131.90,-115.17,-0.00),v40,z0,tcp\WObj:=Plywood;
    MoveL Offs(pOrigin,130.13,-112.13,-0.00),v40,z0,tcp\WObj:=Plywood;
    MoveL Offs(pOrigin,128.61,-110.61,-0.00),v40,z0,tcp\WObj:=Plywood;
    MoveL Offs(pOrigin,126.71,-109.41,-0.00),v40,z0,tcp\WObj:=Plywood;
    MoveL Offs(pOrigin,122.91,-108.14,-0.00),v40,z0,tcp\WObj:=Plywood;
    MoveL Offs(pOrigin,119.11,-108.14,-0.00),v40,z0,tcp\WObj:=Plywood;
    MoveL Offs(pOrigin,117.02,-108.65,-0.00),v40,z0,tcp\WObj:=Plywood;
    MoveL Offs(pOrigin,114.55,-109.79,-0.00),v40,z0,tcp\WObj:=Plywood;
    MoveL Offs(pOrigin,111.70,-112.13,-0.00),v40,z0,tcp\WObj:=Plywood;
    MoveL Offs(pOrigin,110.63,-113.65,-0.00),v40,z0,tcp\WObj:=Plywood;
    MoveL Offs(pOrigin,109.61,-116.12,-0.00),v40,z0,tcp\WObj:=Plywood;
    MoveL Offs(pOrigin,109.23,-117.83,-0.00),v40,fine,tcp\WObj:=Plywood;
    MoveL Offs(pOrigin,109.23,-117.83,-6.00),v60,z5,tcp\WObj:=Plywood;
    MoveL Offs(pOrigin,114.62,-118.78,-6.00),vTravel,z5,tcp\WObj:=Plywood;
    MoveL Offs(pOrigin,114.62,-118.78,-0.00),v60,z0,tcp\WObj:=Plywood;
    MoveL Offs(pOrigin,116.26,-116.50,-0.00),v40,z0,tcp\WObj:=Plywood;
    MoveL Offs(pOrigin,119.11,-114.98,-0.00),v40,z0,tcp\WObj:=Plywood;
    MoveL Offs(pOrigin,122.34,-114.79,-0.00),v40,z0,tcp\WObj:=Plywood;
    MoveL Offs(pOrigin,124.62,-115.93,-0.00),v40,z0,tcp\WObj:=Plywood;
    MoveL Offs(pOrigin,125.76,-117.83,-0.00),v40,z0,tcp\WObj:=Plywood;
    MoveL Offs(pOrigin,125.76,-121.25,-0.00),v40,z0,tcp\WObj:=Plywood;
    MoveL Offs(pOrigin,124.18,-125.61,-0.00),v40,z0,tcp\WObj:=Plywood;
    MoveL Offs(pOrigin,121.64,-129.98,-0.00),v40,z0,tcp\WObj:=Plywood;
    MoveL Offs(pOrigin,117.97,-135.11,-0.00),v40,z0,tcp\WObj:=Plywood;
    MoveL Offs(pOrigin,116.83,-135.81,-0.00),v40,z0,tcp\WObj:=Plywood;
    MoveL Offs(pOrigin,114.55,-127.32,-0.00),v40,z0,tcp\WObj:=Plywood;
    MoveL Offs(pOrigin,113.98,-123.34,-0.00),v40,z0,tcp\WObj:=Plywood;
    MoveL Offs(pOrigin,114.17,-120.30,-0.00),v40,z0,tcp\WObj:=Plywood;
    MoveL Offs(pOrigin,114.62,-118.78,-0.00),v40,fine,tcp\WObj:=Plywood;
    MoveL Offs(pOrigin,114.62,-118.78,-6.00),v60,z5,tcp\WObj:=Plywood;
    MoveL Offs(pOrigin,115.69,-119.92,-6.00),vTravel,z5,tcp\WObj:=Plywood;
    MoveL Offs(pOrigin,115.69,-119.92,-0.00),v60,z0,tcp\WObj:=Plywood;
    MoveL Offs(pOrigin,115.31,-123.15,-0.00),v40,z0,tcp\WObj:=Plywood;
    MoveL Offs(pOrigin,116.26,-129.22,-0.00),v40,z0,tcp\WObj:=Plywood;
    MoveL Offs(pOrigin,117.21,-131.19,-0.00),v40,z0,tcp\WObj:=Plywood;
    MoveL Offs(pOrigin,117.59,-130.74,-0.00),v40,z0,tcp\WObj:=Plywood;
    MoveL Offs(pOrigin,117.59,-128.65,-0.00),v40,z0,tcp\WObj:=Plywood;
    MoveL Offs(pOrigin,116.83,-122.77,-0.00),v40,z0,tcp\WObj:=Plywood;
    MoveL Offs(pOrigin,117.02,-118.97,-0.00),v40,z0,tcp\WObj:=Plywood;
    MoveL Offs(pOrigin,116.45,-118.46,-0.00),v40,z0,tcp\WObj:=Plywood;
    MoveL Offs(pOrigin,115.69,-119.92,-0.00),v40,fine,tcp\WObj:=Plywood;
    MoveL Offs(pOrigin,115.69,-119.92,-6.00),v60,z5,tcp\WObj:=Plywood;
    MoveL Offs(pOrigin,119.87,-104.28,-6.00),vTravel,z5,tcp\WObj:=Plywood;
    MoveL Offs(pOrigin,119.87,-104.28,-0.00),v60,z0,tcp\WObj:=Plywood;
    MoveL Offs(pOrigin,119.49,-104.15,-0.00),v40,z0,tcp\WObj:=Plywood;
    MoveL Offs(pOrigin,119.68,-101.30,-0.00),v40,z0,tcp\WObj:=Plywood;
    MoveL Offs(pOrigin,119.11,-99.97,-0.00),v40,z0,tcp\WObj:=Plywood;
    MoveL Offs(pOrigin,119.24,-98.45,-0.00),v40,z0,tcp\WObj:=Plywood;
    MoveL Offs(pOrigin,120.82,-97.44,-0.00),v40,z0,tcp\WObj:=Plywood;
    MoveL Offs(pOrigin,122.91,-97.06,-0.00),v40,z0,tcp\WObj:=Plywood;
    MoveL Offs(pOrigin,123.54,-95.48,-0.00),v40,z0,tcp\WObj:=Plywood;
    MoveL Offs(pOrigin,123.86,-95.35,-0.00),v40,z0,tcp\WObj:=Plywood;
    MoveL Offs(pOrigin,124.49,-95.60,-0.00),v40,z0,tcp\WObj:=Plywood;
    MoveL Offs(pOrigin,124.62,-97.31,-0.00),v40,z0,tcp\WObj:=Plywood;
    MoveL Offs(pOrigin,126.71,-98.45,-0.00),v40,z0,tcp\WObj:=Plywood;
    MoveL Offs(pOrigin,127.47,-99.59,-0.00),v40,z0,tcp\WObj:=Plywood;
    MoveL Offs(pOrigin,127.34,-100.54,-0.00),v40,z0,tcp\WObj:=Plywood;
    MoveL Offs(pOrigin,126.33,-102.63,-0.00),v40,z0,tcp\WObj:=Plywood;
    MoveL Offs(pOrigin,126.33,-103.96,-0.00),v40,z0,tcp\WObj:=Plywood;
    MoveL Offs(pOrigin,126.71,-104.91,-0.00),v40,z0,tcp\WObj:=Plywood;
    MoveL Offs(pOrigin,126.52,-105.29,-0.00),v40,z0,tcp\WObj:=Plywood;
    MoveL Offs(pOrigin,125.89,-105.10,-0.00),v40,z0,tcp\WObj:=Plywood;
    MoveL Offs(pOrigin,125.38,-103.96,-0.00),v40,z0,tcp\WObj:=Plywood;
    MoveL Offs(pOrigin,125.38,-102.63,-0.00),v40,z0,tcp\WObj:=Plywood;
    MoveL Offs(pOrigin,126.33,-99.97,-0.00),v40,z0,tcp\WObj:=Plywood;
    MoveL Offs(pOrigin,125.00,-98.71,-0.00),v40,z0,tcp\WObj:=Plywood;
    MoveL Offs(pOrigin,124.18,-99.21,-0.00),v40,z0,tcp\WObj:=Plywood;
    MoveL Offs(pOrigin,123.35,-103.39,-0.00),v40,z0,tcp\WObj:=Plywood;
    MoveL Offs(pOrigin,122.91,-103.77,-0.00),v40,z0,tcp\WObj:=Plywood;
    MoveL Offs(pOrigin,122.47,-103.58,-0.00),v40,z0,tcp\WObj:=Plywood;
    MoveL Offs(pOrigin,122.53,-101.30,-0.00),v40,z0,tcp\WObj:=Plywood;
    MoveL Offs(pOrigin,122.91,-99.97,-0.00),v40,z0,tcp\WObj:=Plywood;
    MoveL Offs(pOrigin,122.91,-98.64,-0.00),v40,z0,tcp\WObj:=Plywood;
    MoveL Offs(pOrigin,122.53,-98.26,-0.00),v40,z0,tcp\WObj:=Plywood;
    MoveL Offs(pOrigin,121.39,-98.39,-0.00),v40,z0,tcp\WObj:=Plywood;
    MoveL Offs(pOrigin,120.57,-99.21,-0.00),v40,z0,tcp\WObj:=Plywood;
    MoveL Offs(pOrigin,120.82,-102.63,-0.00),v40,z0,tcp\WObj:=Plywood;
    MoveL Offs(pOrigin,120.44,-103.77,-0.00),v40,z0,tcp\WObj:=Plywood;
    MoveL Offs(pOrigin,119.87,-104.28,-0.00),v40,fine,tcp\WObj:=Plywood;
    MoveL Offs(pOrigin,119.87,-104.28,-6.00),v60,z5,tcp\WObj:=Plywood;
    MoveL Offs(pOrigin,138.93,-106.43,-6.00),vTravel,z5,tcp\WObj:=Plywood;
    MoveL Offs(pOrigin,138.93,-106.43,-0.00),v60,z0,tcp\WObj:=Plywood;
    MoveL Offs(pOrigin,140.07,-104.15,-0.00),v40,z0,tcp\WObj:=Plywood;
    MoveL Offs(pOrigin,141.72,-103.39,-0.00),v40,z0,tcp\WObj:=Plywood;
    MoveL Offs(pOrigin,145.13,-103.71,-0.00),v40,z0,tcp\WObj:=Plywood;
    MoveL Offs(pOrigin,148.17,-103.39,-0.00),v40,z0,tcp\WObj:=Plywood;
    MoveL Offs(pOrigin,151.02,-102.38,-0.00),v40,z0,tcp\WObj:=Plywood;
    MoveL Offs(pOrigin,153.49,-100.80,-0.00),v40,z0,tcp\WObj:=Plywood;
    MoveL Offs(pOrigin,153.87,-100.92,-0.00),v40,z0,tcp\WObj:=Plywood;
    MoveL Offs(pOrigin,151.40,-103.96,-0.00),v40,z0,tcp\WObj:=Plywood;
    MoveL Offs(pOrigin,147.79,-106.49,-0.00),v40,z0,tcp\WObj:=Plywood;
    MoveL Offs(pOrigin,145.32,-107.19,-0.00),v40,z0,tcp\WObj:=Plywood;
    MoveL Offs(pOrigin,142.09,-107.19,-0.00),v40,z0,tcp\WObj:=Plywood;
    MoveL Offs(pOrigin,138.93,-106.43,-0.00),v40,fine,tcp\WObj:=Plywood;
    MoveL Offs(pOrigin,138.93,-106.43,-6.00),v60,z5,tcp\WObj:=Plywood;
    MoveL Offs(pOrigin,139.82,-118.59,-6.00),vTravel,z5,tcp\WObj:=Plywood;
    MoveL Offs(pOrigin,139.82,-118.59,-0.00),v60,z0,tcp\WObj:=Plywood;
    MoveL Offs(pOrigin,133.74,-118.84,-0.00),v40,z0,tcp\WObj:=Plywood;
    MoveL Offs(pOrigin,133.36,-119.54,-0.00),v40,z0,tcp\WObj:=Plywood;
    MoveL Offs(pOrigin,132.98,-123.34,-0.00),v40,z0,tcp\WObj:=Plywood;
    MoveL Offs(pOrigin,131.52,-127.32,-0.00),v40,z0,tcp\WObj:=Plywood;
    MoveL Offs(pOrigin,127.34,-133.78,-0.00),v40,z0,tcp\WObj:=Plywood;
    MoveL Offs(pOrigin,129.37,-134.16,-0.00),v40,z0,tcp\WObj:=Plywood;
    MoveL Offs(pOrigin,137.16,-134.16,-0.00),v40,z0,tcp\WObj:=Plywood;
    MoveL Offs(pOrigin,145.70,-133.40,-0.00),v40,z0,tcp\WObj:=Plywood;
    MoveL Offs(pOrigin,156.53,-130.93,-0.00),v40,z0,tcp\WObj:=Plywood;
    MoveL Offs(pOrigin,160.52,-129.16,-0.00),v40,z0,tcp\WObj:=Plywood;
    MoveL Offs(pOrigin,161.60,-128.27,-0.00),v40,z0,tcp\WObj:=Plywood;
    MoveL Offs(pOrigin,161.66,-126.94,-0.00),v40,z0,tcp\WObj:=Plywood;
    MoveL Offs(pOrigin,160.08,-114.60,-0.00),v40,z0,tcp\WObj:=Plywood;
    MoveL Offs(pOrigin,159.57,-114.22,-0.00),v40,z0,tcp\WObj:=Plywood;
    MoveL Offs(pOrigin,155.96,-115.74,-0.00),v40,z0,tcp\WObj:=Plywood;
  ENDPROC

  PROC DrawPart6()
    MoveL Offs(pOrigin,147.03,-117.64,-0.00),v40,z0,tcp\WObj:=Plywood;
    MoveL Offs(pOrigin,139.82,-118.59,-0.00),v40,fine,tcp\WObj:=Plywood;
    MoveL Offs(pOrigin,139.82,-118.59,-6.00),v60,z5,tcp\WObj:=Plywood;
    MoveL Offs(pOrigin,161.03,-109.66,-6.00),vTravel,z5,tcp\WObj:=Plywood;
    MoveL Offs(pOrigin,161.03,-109.66,-0.00),v60,z0,tcp\WObj:=Plywood;
    MoveL Offs(pOrigin,162.99,-112.51,-0.00),v40,z0,tcp\WObj:=Plywood;
    MoveL Offs(pOrigin,165.65,-114.98,-0.00),v40,z0,tcp\WObj:=Plywood;
    MoveL Offs(pOrigin,168.31,-116.62,-0.00),v40,z0,tcp\WObj:=Plywood;
    MoveL Offs(pOrigin,173.25,-118.59,-0.00),v40,z0,tcp\WObj:=Plywood;
    MoveL Offs(pOrigin,179.89,-119.92,-0.00),v40,z0,tcp\WObj:=Plywood;
    MoveL Offs(pOrigin,185.97,-120.11,-0.00),v40,z0,tcp\WObj:=Plywood;
    MoveL Offs(pOrigin,191.29,-119.16,-0.00),v40,z0,tcp\WObj:=Plywood;
    MoveL Offs(pOrigin,194.14,-118.08,-0.00),v40,z0,tcp\WObj:=Plywood;
    MoveL Offs(pOrigin,197.56,-116.37,-0.00),v40,z0,tcp\WObj:=Plywood;
    MoveL Offs(pOrigin,200.22,-114.60,-0.00),v40,z0,tcp\WObj:=Plywood;
    MoveL Offs(pOrigin,204.02,-110.99,-0.00),v40,z0,tcp\WObj:=Plywood;
    MoveL Offs(pOrigin,204.97,-109.66,-0.00),v40,z0,tcp\WObj:=Plywood;
    MoveL Offs(pOrigin,204.78,-109.28,-0.00),v40,z0,tcp\WObj:=Plywood;
    MoveL Offs(pOrigin,202.88,-108.46,-0.00),v40,z0,tcp\WObj:=Plywood;
    MoveL Offs(pOrigin,201.55,-107.38,-0.00),v40,z0,tcp\WObj:=Plywood;
    MoveL Offs(pOrigin,199.20,-103.96,-0.00),v40,z0,tcp\WObj:=Plywood;
    MoveL Offs(pOrigin,198.13,-100.54,-0.00),v40,z0,tcp\WObj:=Plywood;
    MoveL Offs(pOrigin,196.23,-87.63,-0.00),v40,z0,tcp\WObj:=Plywood;
    MoveL Offs(pOrigin,195.15,-84.02,-0.00),v40,z0,tcp\WObj:=Plywood;
    MoveL Offs(pOrigin,193.32,-79.65,-0.00),v40,z0,tcp\WObj:=Plywood;
    MoveL Offs(pOrigin,191.35,-76.23,-0.00),v40,z0,tcp\WObj:=Plywood;
    MoveL Offs(pOrigin,188.44,-72.24,-0.00),v40,z0,tcp\WObj:=Plywood;
    MoveL Offs(pOrigin,185.21,-69.20,-0.00),v40,z0,tcp\WObj:=Plywood;
    MoveL Offs(pOrigin,181.60,-66.86,-0.00),v40,z0,tcp\WObj:=Plywood;
    MoveL Offs(pOrigin,177.99,-65.40,-0.00),v40,z0,tcp\WObj:=Plywood;
    MoveL Offs(pOrigin,175.34,-64.83,-0.00),v40,z0,tcp\WObj:=Plywood;
    MoveL Offs(pOrigin,171.92,-64.83,-0.00),v40,z0,tcp\WObj:=Plywood;
    MoveL Offs(pOrigin,169.45,-65.40,-0.00),v40,z0,tcp\WObj:=Plywood;
    MoveL Offs(pOrigin,166.98,-66.42,-0.00),v40,z0,tcp\WObj:=Plywood;
    MoveL Offs(pOrigin,164.07,-68.63,-0.00),v40,z0,tcp\WObj:=Plywood;
    MoveL Offs(pOrigin,165.77,-72.62,-0.00),v40,z0,tcp\WObj:=Plywood;
    MoveL Offs(pOrigin,166.79,-76.23,-0.00),v40,z0,tcp\WObj:=Plywood;
    MoveL Offs(pOrigin,166.98,-79.27,-0.00),v40,z0,tcp\WObj:=Plywood;
    MoveL Offs(pOrigin,166.79,-83.45,-0.00),v40,z0,tcp\WObj:=Plywood;
    MoveL Offs(pOrigin,166.22,-86.11,-0.00),v40,z0,tcp\WObj:=Plywood;
    MoveL Offs(pOrigin,163.12,-93.89,-0.00),v40,z0,tcp\WObj:=Plywood;
    MoveL Offs(pOrigin,164.70,-96.74,-0.00),v40,z0,tcp\WObj:=Plywood;
    MoveL Offs(pOrigin,165.08,-97.06,-0.00),v40,z0,tcp\WObj:=Plywood;
    MoveL Offs(pOrigin,165.58,-96.81,-0.00),v40,z0,tcp\WObj:=Plywood;
    MoveL Offs(pOrigin,165.65,-98.26,-0.00),v40,z0,tcp\WObj:=Plywood;
    MoveL Offs(pOrigin,170.02,-103.01,-0.00),v40,z0,tcp\WObj:=Plywood;
    MoveL Offs(pOrigin,172.68,-105.10,-0.00),v40,z0,tcp\WObj:=Plywood;
    MoveL Offs(pOrigin,178.37,-108.46,-0.00),v40,z0,tcp\WObj:=Plywood;
    MoveL Offs(pOrigin,180.65,-109.34,-0.00),v40,z0,tcp\WObj:=Plywood;
    MoveL Offs(pOrigin,187.68,-110.80,-0.00),v40,z0,tcp\WObj:=Plywood;
    MoveL Offs(pOrigin,192.43,-110.80,-0.00),v40,z0,tcp\WObj:=Plywood;
    MoveL Offs(pOrigin,198.89,-109.72,-0.00),v40,z0,tcp\WObj:=Plywood;
    MoveL Offs(pOrigin,199.39,-110.04,-0.00),v40,z0,tcp\WObj:=Plywood;
    MoveL Offs(pOrigin,198.89,-110.42,-0.00),v40,z0,tcp\WObj:=Plywood;
    MoveL Offs(pOrigin,194.52,-111.37,-0.00),v40,z0,tcp\WObj:=Plywood;
    MoveL Offs(pOrigin,188.25,-111.94,-0.00),v40,z0,tcp\WObj:=Plywood;
    MoveL Offs(pOrigin,183.88,-111.37,-0.00),v40,z0,tcp\WObj:=Plywood;
    MoveL Offs(pOrigin,178.75,-109.72,-0.00),v40,z0,tcp\WObj:=Plywood;
    MoveL Offs(pOrigin,175.34,-108.01,-0.00),v40,z0,tcp\WObj:=Plywood;
    MoveL Offs(pOrigin,170.02,-104.34,-0.00),v40,z0,tcp\WObj:=Plywood;
    MoveL Offs(pOrigin,165.65,-99.97,-0.00),v40,z0,tcp\WObj:=Plywood;
    MoveL Offs(pOrigin,162.42,-95.73,-0.00),v40,z0,tcp\WObj:=Plywood;
    MoveL Offs(pOrigin,161.91,-96.17,-0.00),v40,z0,tcp\WObj:=Plywood;
    MoveL Offs(pOrigin,160.90,-98.83,-0.00),v40,z0,tcp\WObj:=Plywood;
    MoveL Offs(pOrigin,159.95,-103.39,-0.00),v40,z0,tcp\WObj:=Plywood;
    MoveL Offs(pOrigin,159.95,-107.19,-0.00),v40,z0,tcp\WObj:=Plywood;
    MoveL Offs(pOrigin,161.03,-109.66,-0.00),v40,fine,tcp\WObj:=Plywood;
    MoveL Offs(pOrigin,161.03,-109.66,-6.00),v60,z5,tcp\WObj:=Plywood;
    MoveL Offs(pOrigin,167.36,-99.15,-6.00),vTravel,z5,tcp\WObj:=Plywood;
    MoveL Offs(pOrigin,167.36,-99.15,-0.00),v60,z0,tcp\WObj:=Plywood;
    MoveL Offs(pOrigin,166.79,-98.39,-0.00),v40,z0,tcp\WObj:=Plywood;
    MoveL Offs(pOrigin,167.48,-98.45,-0.00),v40,z0,tcp\WObj:=Plywood;
    MoveL Offs(pOrigin,167.36,-99.15,-0.00),v40,fine,tcp\WObj:=Plywood;
    MoveL Offs(pOrigin,167.36,-99.15,-6.00),v60,z5,tcp\WObj:=Plywood;
    MoveL Offs(pOrigin,151.59,-91.42,-6.00),vTravel,z5,tcp\WObj:=Plywood;
    MoveL Offs(pOrigin,151.59,-91.42,-0.00),v60,z0,tcp\WObj:=Plywood;
    MoveL Offs(pOrigin,149.88,-92.82,-0.00),v40,z0,tcp\WObj:=Plywood;
    MoveL Offs(pOrigin,146.46,-93.70,-0.00),v40,z0,tcp\WObj:=Plywood;
    MoveL Offs(pOrigin,143.61,-93.32,-0.00),v40,z0,tcp\WObj:=Plywood;
    MoveL Offs(pOrigin,141.34,-92.25,-0.00),v40,z0,tcp\WObj:=Plywood;
    MoveL Offs(pOrigin,139.63,-90.85,-0.00),v40,z0,tcp\WObj:=Plywood;
    MoveL Offs(pOrigin,138.42,-88.96,-0.00),v40,z0,tcp\WObj:=Plywood;
    MoveL Offs(pOrigin,138.11,-86.30,-0.00),v40,z0,tcp\WObj:=Plywood;
    MoveL Offs(pOrigin,138.30,-85.92,-0.00),v40,z0,tcp\WObj:=Plywood;
    MoveL Offs(pOrigin,138.87,-85.79,-0.00),v40,z0,tcp\WObj:=Plywood;
    MoveL Offs(pOrigin,142.09,-88.26,-0.00),v40,z0,tcp\WObj:=Plywood;
    MoveL Offs(pOrigin,145.51,-89.34,-0.00),v40,z0,tcp\WObj:=Plywood;
    MoveL Offs(pOrigin,148.17,-89.15,-0.00),v40,z0,tcp\WObj:=Plywood;
    MoveL Offs(pOrigin,151.97,-87.50,-0.00),v40,z0,tcp\WObj:=Plywood;
    MoveL Offs(pOrigin,152.54,-88.58,-0.00),v40,z0,tcp\WObj:=Plywood;
    MoveL Offs(pOrigin,152.54,-89.53,-0.00),v40,z0,tcp\WObj:=Plywood;
    MoveL Offs(pOrigin,151.59,-91.42,-0.00),v40,fine,tcp\WObj:=Plywood;
    MoveL Offs(pOrigin,151.59,-91.42,-6.00),v60,z5,tcp\WObj:=Plywood;
    MoveL Offs(pOrigin,161.09,-65.02,-6.00),vTravel,z5,tcp\WObj:=Plywood;
    MoveL Offs(pOrigin,161.09,-65.02,-0.00),v60,z0,tcp\WObj:=Plywood;
    MoveL Offs(pOrigin,161.85,-65.21,-0.00),v40,z0,tcp\WObj:=Plywood;
    MoveL Offs(pOrigin,167.36,-62.24,-0.00),v40,z0,tcp\WObj:=Plywood;
    MoveL Offs(pOrigin,172.11,-58.56,-0.00),v40,z0,tcp\WObj:=Plywood;
    MoveL Offs(pOrigin,175.53,-54.77,-0.00),v40,z0,tcp\WObj:=Plywood;
    MoveL Offs(pOrigin,177.55,-51.54,-0.00),v40,z0,tcp\WObj:=Plywood;
    MoveL Offs(pOrigin,178.56,-49.26,-0.00),v40,z0,tcp\WObj:=Plywood;
    MoveL Offs(pOrigin,177.80,-48.69,-0.00),v40,z0,tcp\WObj:=Plywood;
    MoveL Offs(pOrigin,172.68,-48.81,-0.00),v40,z0,tcp\WObj:=Plywood;
    MoveL Offs(pOrigin,170.59,-52.11,-0.00),v40,z0,tcp\WObj:=Plywood;
    MoveL Offs(pOrigin,168.88,-53.31,-0.00),v40,z0,tcp\WObj:=Plywood;
    MoveL Offs(pOrigin,166.22,-54.39,-0.00),v40,z0,tcp\WObj:=Plywood;
    MoveL Offs(pOrigin,163.75,-54.96,-0.00),v40,z0,tcp\WObj:=Plywood;
    MoveL Offs(pOrigin,155.20,-55.15,-0.00),v40,z0,tcp\WObj:=Plywood;
    MoveL Offs(pOrigin,151.02,-55.91,-0.00),v40,z0,tcp\WObj:=Plywood;
    MoveL Offs(pOrigin,149.44,-56.66,-0.00),v40,z0,tcp\WObj:=Plywood;
    MoveL Offs(pOrigin,156.15,-60.46,-0.00),v40,z0,tcp\WObj:=Plywood;
    MoveL Offs(pOrigin,159.38,-63.12,-0.00),v40,z0,tcp\WObj:=Plywood;
    MoveL Offs(pOrigin,161.09,-65.02,-0.00),v40,fine,tcp\WObj:=Plywood;
    MoveL Offs(pOrigin,161.09,-65.02,-6.00),v60,z5,tcp\WObj:=Plywood;
    MoveL Offs(pOrigin,116.45,-48.12,-6.00),vTravel,z5,tcp\WObj:=Plywood;
    MoveL Offs(pOrigin,116.45,-48.12,-0.00),v60,z0,tcp\WObj:=Plywood;
    MoveL Offs(pOrigin,116.45,-45.84,-0.00),v40,z0,tcp\WObj:=Plywood;
    MoveL Offs(pOrigin,115.95,-44.51,-0.00),v40,z0,tcp\WObj:=Plywood;
    MoveL Offs(pOrigin,114.93,-43.50,-0.00),v40,z0,tcp\WObj:=Plywood;
    MoveL Offs(pOrigin,113.41,-42.99,-0.00),v40,z0,tcp\WObj:=Plywood;
  ENDPROC

  PROC DrawPart7()
    MoveL Offs(pOrigin,112.27,-43.56,-0.00),v40,z0,tcp\WObj:=Plywood;
    MoveL Offs(pOrigin,111.45,-44.51,-0.00),v40,z0,tcp\WObj:=Plywood;
    MoveL Offs(pOrigin,109.99,-47.55,-0.00),v40,z0,tcp\WObj:=Plywood;
    MoveL Offs(pOrigin,109.61,-47.17,-0.00),v40,z0,tcp\WObj:=Plywood;
    MoveL Offs(pOrigin,109.42,-45.27,-0.00),v40,z0,tcp\WObj:=Plywood;
    MoveL Offs(pOrigin,108.92,-43.94,-0.00),v40,z0,tcp\WObj:=Plywood;
    MoveL Offs(pOrigin,108.09,-42.86,-0.00),v40,z0,tcp\WObj:=Plywood;
    MoveL Offs(pOrigin,106.77,-42.04,-0.00),v40,z0,tcp\WObj:=Plywood;
    MoveL Offs(pOrigin,105.63,-42.04,-0.00),v40,z0,tcp\WObj:=Plywood;
    MoveL Offs(pOrigin,104.87,-42.42,-0.00),v40,z0,tcp\WObj:=Plywood;
    MoveL Offs(pOrigin,103.98,-43.56,-0.00),v40,z0,tcp\WObj:=Plywood;
    MoveL Offs(pOrigin,103.28,-45.46,-0.00),v40,z0,tcp\WObj:=Plywood;
    MoveL Offs(pOrigin,102.78,-45.84,-0.00),v40,z0,tcp\WObj:=Plywood;
    MoveL Offs(pOrigin,102.46,-45.65,-0.00),v40,z0,tcp\WObj:=Plywood;
    MoveL Offs(pOrigin,102.08,-43.75,-0.00),v40,z0,tcp\WObj:=Plywood;
    MoveL Offs(pOrigin,101.45,-42.61,-0.00),v40,z0,tcp\WObj:=Plywood;
    MoveL Offs(pOrigin,100.50,-41.79,-0.00),v40,z0,tcp\WObj:=Plywood;
    MoveL Offs(pOrigin,99.36,-41.41,-0.00),v40,z0,tcp\WObj:=Plywood;
    MoveL Offs(pOrigin,97.84,-41.72,-0.00),v40,z0,tcp\WObj:=Plywood;
    MoveL Offs(pOrigin,96.70,-42.61,-0.00),v40,z0,tcp\WObj:=Plywood;
    MoveL Offs(pOrigin,95.18,-45.65,-0.00),v40,z0,tcp\WObj:=Plywood;
    MoveL Offs(pOrigin,94.23,-43.18,-0.00),v40,z0,tcp\WObj:=Plywood;
    MoveL Offs(pOrigin,92.71,-42.23,-0.00),v40,z0,tcp\WObj:=Plywood;
    MoveL Offs(pOrigin,91.57,-42.36,-0.00),v40,z0,tcp\WObj:=Plywood;
    MoveL Offs(pOrigin,90.24,-43.37,-0.00),v40,z0,tcp\WObj:=Plywood;
    MoveL Offs(pOrigin,89.86,-44.13,-0.00),v40,z0,tcp\WObj:=Plywood;
    MoveL Offs(pOrigin,89.86,-45.46,-0.00),v40,z0,tcp\WObj:=Plywood;
    MoveL Offs(pOrigin,90.75,-48.50,-0.00),v40,z0,tcp\WObj:=Plywood;
    MoveL Offs(pOrigin,92.90,-52.11,-0.00),v40,z0,tcp\WObj:=Plywood;
    MoveL Offs(pOrigin,95.56,-54.77,-0.00),v40,z0,tcp\WObj:=Plywood;
    MoveL Offs(pOrigin,97.65,-56.16,-0.00),v40,z0,tcp\WObj:=Plywood;
    MoveL Offs(pOrigin,102.02,-57.80,-0.00),v40,z0,tcp\WObj:=Plywood;
    MoveL Offs(pOrigin,106.39,-57.80,-0.00),v40,z0,tcp\WObj:=Plywood;
    MoveL Offs(pOrigin,109.61,-56.73,-0.00),v40,z0,tcp\WObj:=Plywood;
    MoveL Offs(pOrigin,111.89,-55.34,-0.00),v40,z0,tcp\WObj:=Plywood;
    MoveL Offs(pOrigin,113.41,-54.01,-0.00),v40,z0,tcp\WObj:=Plywood;
    MoveL Offs(pOrigin,115.00,-51.92,-0.00),v40,z0,tcp\WObj:=Plywood;
    MoveL Offs(pOrigin,116.45,-48.12,-0.00),v40,fine,tcp\WObj:=Plywood;
    MoveL Offs(pOrigin,116.45,-48.12,-6.00),v60,z5,tcp\WObj:=Plywood;
    MoveL Offs(pOrigin,98.79,-146.45,-6.00),vTravel,z5,tcp\WObj:=Plywood;
    MoveL Offs(pOrigin,98.79,-146.45,-0.00),v60,z0,tcp\WObj:=Plywood;
    MoveL Offs(pOrigin,98.22,-146.70,-0.00),v40,z0,tcp\WObj:=Plywood;
    MoveL Offs(pOrigin,97.84,-147.65,-0.00),v40,z0,tcp\WObj:=Plywood;
    MoveL Offs(pOrigin,97.84,-151.45,-0.00),v40,z0,tcp\WObj:=Plywood;
    MoveL Offs(pOrigin,98.34,-153.16,-0.00),v40,z0,tcp\WObj:=Plywood;
    MoveL Offs(pOrigin,99.93,-156.20,-0.00),v40,z0,tcp\WObj:=Plywood;
    MoveL Offs(pOrigin,102.02,-158.47,-0.00),v40,z0,tcp\WObj:=Plywood;
    MoveL Offs(pOrigin,104.87,-160.44,-0.00),v40,z0,tcp\WObj:=Plywood;
    MoveL Offs(pOrigin,109.42,-162.27,-0.00),v40,z0,tcp\WObj:=Plywood;
    MoveL Offs(pOrigin,114.55,-163.03,-0.00),v40,z0,tcp\WObj:=Plywood;
    MoveL Offs(pOrigin,117.02,-163.03,-0.00),v40,z0,tcp\WObj:=Plywood;
    MoveL Offs(pOrigin,121.58,-162.15,-0.00),v40,z0,tcp\WObj:=Plywood;
    MoveL Offs(pOrigin,123.67,-161.26,-0.00),v40,z0,tcp\WObj:=Plywood;
    MoveL Offs(pOrigin,126.14,-159.61,-0.00),v40,z0,tcp\WObj:=Plywood;
    MoveL Offs(pOrigin,128.61,-156.96,-0.00),v40,z0,tcp\WObj:=Plywood;
    MoveL Offs(pOrigin,129.75,-154.87,-0.00),v40,z0,tcp\WObj:=Plywood;
    MoveL Offs(pOrigin,129.56,-154.55,-0.00),v40,z0,tcp\WObj:=Plywood;
    MoveL Offs(pOrigin,119.49,-153.73,-0.00),v40,z0,tcp\WObj:=Plywood;
    MoveL Offs(pOrigin,112.46,-152.21,-0.00),v40,z0,tcp\WObj:=Plywood;
    MoveL Offs(pOrigin,102.21,-148.47,-0.00),v40,z0,tcp\WObj:=Plywood;
    MoveL Offs(pOrigin,98.79,-146.45,-0.00),v40,fine,tcp\WObj:=Plywood;
    MoveL Offs(pOrigin,98.79,-146.45,-6.00),v60,z5,tcp\WObj:=Plywood;
    MoveL Offs(pOrigin,105.25,-162.34,-6.00),vTravel,z5,tcp\WObj:=Plywood;
    MoveL Offs(pOrigin,105.25,-162.34,-0.00),v60,z0,tcp\WObj:=Plywood;
    MoveL Offs(pOrigin,105.12,-162.65,-0.00),v40,z0,tcp\WObj:=Plywood;
    MoveL Offs(pOrigin,106.58,-166.45,-0.00),v40,z0,tcp\WObj:=Plywood;
    MoveL Offs(pOrigin,108.16,-172.34,-0.00),v40,z0,tcp\WObj:=Plywood;
    MoveL Offs(pOrigin,108.47,-172.47,-0.00),v40,z0,tcp\WObj:=Plywood;
    MoveL Offs(pOrigin,115.50,-165.69,-0.00),v40,z0,tcp\WObj:=Plywood;
    MoveL Offs(pOrigin,116.39,-164.36,-0.00),v40,z0,tcp\WObj:=Plywood;
    MoveL Offs(pOrigin,112.27,-163.98,-0.00),v40,z0,tcp\WObj:=Plywood;
    MoveL Offs(pOrigin,105.25,-162.34,-0.00),v40,fine,tcp\WObj:=Plywood;
    MoveL Offs(pOrigin,105.25,-162.34,-6.00),v60,z5,tcp\WObj:=Plywood;
  ENDPROC

ENDMODULE
